(* IEC 61131-3 sources: Industry-PLC-LLM/data/PLCBEAD_repo/PLCBEAD_PLCEmbed-main/PLC-BEAD/Source/GEB/TIME_TO_INT, 1 file *)

(* ---- TIME_TO_INT.ST ---- *)
FUNCTION TIME_TO_INT1:INT

VAR_INPUT
	IN :	TIME;
END_VAR

TIME_TO_INT1 := DINT_TO_INT(TIME_TO_DINT(IN));
END_FUNCTION

PROGRAM program0
  VAR
	IN :	TIME;
    CEIL5_OUT : INT;
  END_VAR

  CEIL5_OUT := TIME_TO_INT1(IN);
END_PROGRAM
